# EPICS autosave request: TWINCAT/iocBoot/iocTWINCAT-IOC-01/TWINCAT_01_settings.req
# Motor settings
file "motor_settings.req" P=$(P), M=MTR$(MTRCTRL)01
file "motor_settings.req" P=$(P), M=MTR$(MTRCTRL)02
file "motor_settings.req" P=$(P), M=MTR$(MTRCTRL)03
file "motor_settings.req" P=$(P), M=MTR$(MTRCTRL)04
file "motor_settings.req" P=$(P), M=MTR$(MTRCTRL)05
file "motor_settings.req" P=$(P), M=MTR$(MTRCTRL)06
file "motor_settings.req" P=$(P), M=MTR$(MTRCTRL)07
file "motor_settings.req" P=$(P), M=MTR$(MTRCTRL)08
